// TIA Portal V16 export
// export: Created 2022-02-11T10:36:49.9262593Z, ExportSetting WithDefaults, DisplayName Totally Integrated Automation Portal, DisplayVersion V16 Update 5, DisplayName TIA Portal Version Control Interface, DisplayVersion V16 Update 2, DisplayName TIA Portal Openness, DisplayVersion V16 Update 5, DisplayName STEP 7 Professional, DisplayVersion V16 Update 5, DisplayName STEP 7 Safety, DisplayVersion V16, DisplayName WinCC Professional, DisplayVersion V16 Update 5, DisplayName SIMATIC Visualization Architect, DisplayVersion V16
FUNCTION_BLOCK "fbObjMotor_KM"   // FB9202, LAD
{ S7_Optimized_Access := 'TRUE' }
VERSION : 0.1
// stored: AutoNumber false, IsIECCheckEnabled false, IsRetainMemResEnabled false, MemoryReserve 0, SetENOAutomatically false, UDAEnableTagReadback false
   VAR_INPUT
      aMarxaAuto : Bool := FALSE;   // Activar element mode automatic
      eErrorProteccio : Bool;   // Entrada error proteccio motor filtre
      eConfirmacioMarxa : Bool;   // Senyal confirmacio marxa filtre
      bCM_Marxa : Bool := TRUE;   // Condicions necesaries activar element
      tAla_ConMar : Time := t#3s;   // Temps retard activacio alarma confirmacio marxa
      tAla_CM_Marxa : Time := t#2s;   // Temps retard activacio alarma condicions moviment
      psEnaAutoGrl : "boto";
      psEnaManualGrl : "boto";
      psAnuConMov : Bool;
      psResetAlarma : Bool;
      mFirstScan : Bool;
      "Clock_0.5Hz" : Bool;
      bSysOk : Bool := FALSE;
   END_VAR
   VAR_OUTPUT
      aMarxa : Bool;   // Sortida activacio Filtre
      be_Marxa : Bool;   // Bit estat Marxa (Confirmacio + Proteccio + Sortida)
      be_Parat : Bool;
      al_Proteccio : Bool;   // Alarma proteccio motor
      al_CM_Marxa : Bool;   // Alarma condicions moviment obrir
      al_Marxa : Bool;   // Alarma confirmacio marxa filtre
   END_VAR
   VAR
      psManMarxa : Bool;
      be_Marxa_Err : Bool;   // Error en validacio Confirmacio Marxa. Sense retard per alarma.
      bErrorCM : Bool;   // Error CM. Si activem sortida i no es compleixen les CM. Sense retard
      timAla_CM_Marxa { S7_SetPoint := 'True'} : IEC_TIMER;   // Timer retard alarma condicions moviment
      timAla_Marxa { S7_SetPoint := 'True'} : IEC_TIMER;   // Timer retard alarma marxa filtre
      bCM_Ok { S7_SetPoint := 'True'} : Bool;
      aMarxaSenseTestCM : Bool;   // Bit activacio sortida sense tenir en compte condicions moviment
      mAuxTimer : Bool;   // Bit auxiliarInicialitzacio timers
      HMI : "HMI_oMotor";
      bLast_Alarmes { S7_SetPoint := 'True'} : Bool;
   END_VAR
   VAR_TEMP
      ModeManual : Bool;
      ModeAutomatic : Bool;
      ResetAlarmes : Bool;
   END_VAR
   VAR CONSTANT
      STATUS_OBJ_ERR : Int := 10;
      STATUS_OBJ_WARNING : Int := 11;
      STATUS_OBJ_ON : Int := 1;
      STATUS_OBJ_OFF : Int := 0;
      STATUS_OBJ_UNKNOWN : Int := -1;
   END_VAR
   VAR_TEMP   // added for the SCL form of the ladder/FBD networks
      _w1 : Bool;
   END_VAR
BEGIN

REGION Network 1 (SCL): Descripció
   // Motor activat per Rele, amb confirmacio i proteccio.
END_REGION

REGION Network 2: Test habilitació mode manual. Desactivar si no tenim habilitació manual.
   // psEnaManualGrl : és el pulsador de manual de Appinfo. Si aquest està activar tots els objectes del cicle es troben en Mode Manual.
   // 
   // HMI.psEnaManual : és el pulsador de manual únic de l'objecte. Significa que la resta d'objectes es trobaràn en automàtic menys aquest.
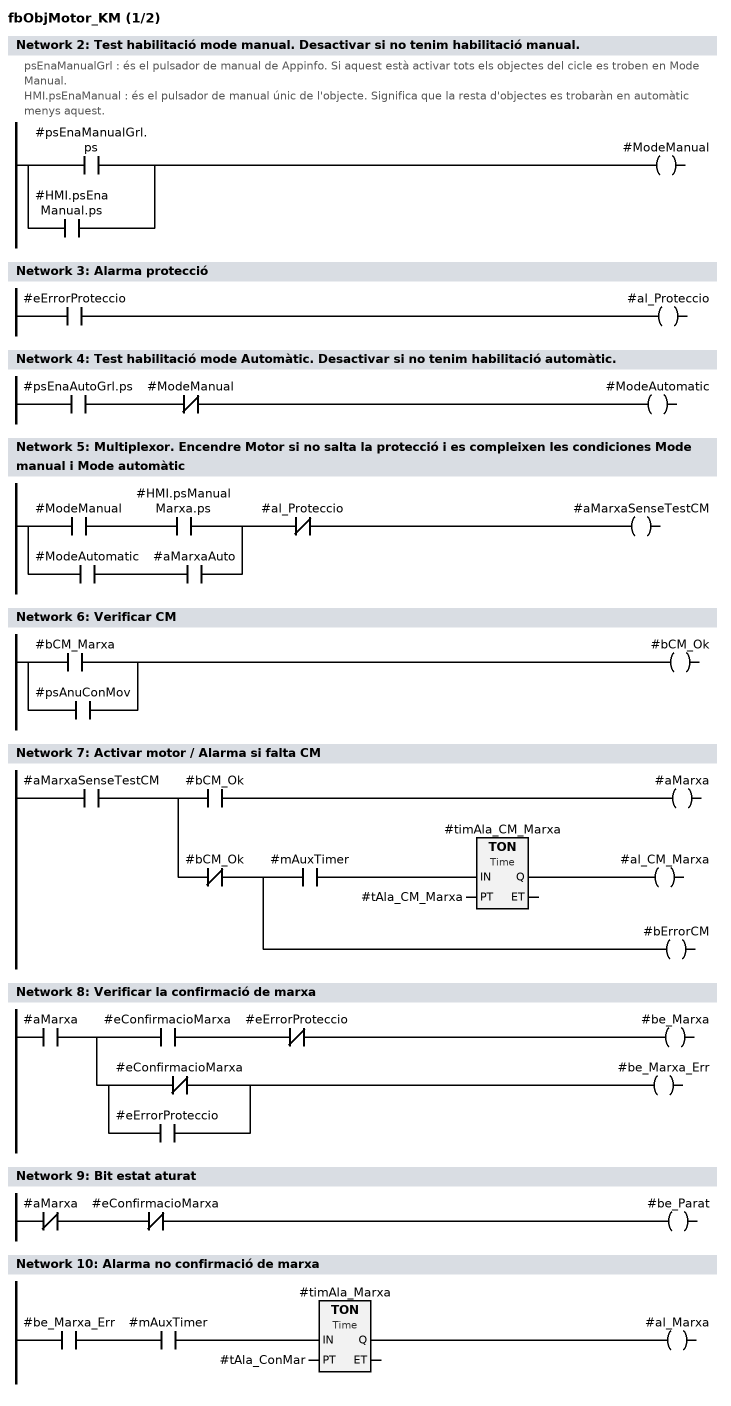
   RUNG wire#powerrail
      Contact( #psEnaManualGrl.ps )
      wire#w1
      Coil( #ModeManual )
   END_RUNG
   RUNG wire#powerrail
      Contact( #HMI.psEnaManual.ps )
   END_RUNG wire#w1
   // the same network as SCL:
   #ModeManual := #psEnaManualGrl.ps OR #HMI.psEnaManual.ps;
END_REGION

REGION Network 3: Alarma protecció
   RUNG wire#powerrail
      Contact( #eErrorProteccio )
      Coil( #al_Proteccio )
   END_RUNG
   // the same network as SCL:
   #al_Proteccio := #eErrorProteccio;
END_REGION

REGION Network 4: Test habilitació mode Automàtic. Desactivar si no tenim habilitació automàtic.
   RUNG wire#powerrail
      Contact( #psEnaAutoGrl.ps )
      I_Contact( #ModeManual )
      Coil( #ModeAutomatic )
   END_RUNG
   // the same network as SCL:
   #ModeAutomatic := #psEnaAutoGrl.ps AND NOT #ModeManual;
END_REGION

REGION Network 5: Multiplexor. Encendre Motor si no salta la protecció i es compleixen les condiciones Mode manual i Mode automàtic
   RUNG wire#powerrail
      Contact( #ModeManual )
      Contact( #HMI.psManualMarxa.ps )
      wire#w1
      I_Contact( #al_Proteccio )
      Coil( #aMarxaSenseTestCM )
   END_RUNG
   RUNG wire#powerrail
      Contact( #ModeAutomatic )
      Contact( #aMarxaAuto )
   END_RUNG wire#w1
   // the same network as SCL:
   #aMarxaSenseTestCM := ((#ModeManual AND #HMI.psManualMarxa.ps) OR (#ModeAutomatic AND #aMarxaAuto)) AND NOT #al_Proteccio;
END_REGION

REGION Network 6: Verificar CM
   RUNG wire#powerrail
      Contact( #bCM_Marxa )
      wire#w1
      Coil( #bCM_Ok )
   END_RUNG
   RUNG wire#powerrail
      Contact( #psAnuConMov )
   END_RUNG wire#w1
   // the same network as SCL:
   #bCM_Ok := #bCM_Marxa OR #psAnuConMov;
END_REGION

REGION Network 7: Activar motor / Alarma si falta CM
   RUNG wire#powerrail
      Contact( #aMarxaSenseTestCM )
      wire#w1
      Contact( #bCM_Ok )
      Coil( #aMarxa )
   END_RUNG
   RUNG wire#w1
      I_Contact( #bCM_Ok )
      wire#w2
      Contact( #mAuxTimer )
      { S7_Templates := "time_type := Time" } #timAla_CM_Marxa.TON(pt := #tAla_CM_Marxa, et =>)
      Coil( #al_CM_Marxa )
   END_RUNG
   RUNG wire#w2
      Coil( #bErrorCM )
   END_RUNG
   // the same network as SCL:
   #aMarxa := #aMarxaSenseTestCM AND #bCM_Ok;
   #_w1 := #aMarxaSenseTestCM AND NOT #bCM_Ok;
   #timAla_CM_Marxa.TON(IN := #_w1 AND #mAuxTimer, PT := #tAla_CM_Marxa);
   #al_CM_Marxa := #timAla_CM_Marxa.Q;
   #bErrorCM := #_w1;
END_REGION

REGION Network 8: Verificar la confirmació de marxa
   RUNG wire#powerrail
      Contact( #aMarxa )
      wire#w1
      Contact( #eConfirmacioMarxa )
      I_Contact( #eErrorProteccio )
      Coil( #be_Marxa )
   END_RUNG
   RUNG wire#w1
      I_Contact( #eConfirmacioMarxa )
      wire#w2
      Coil( #be_Marxa_Err )
   END_RUNG
   RUNG wire#w1
      Contact( #eErrorProteccio )
   END_RUNG wire#w2
   // the same network as SCL:
   #be_Marxa := #aMarxa AND #eConfirmacioMarxa AND NOT #eErrorProteccio;
   #be_Marxa_Err := #aMarxa AND (NOT #eConfirmacioMarxa OR #eErrorProteccio);
END_REGION

REGION Network 9: Bit estat aturat
   RUNG wire#powerrail
      I_Contact( #aMarxa )
      I_Contact( #eConfirmacioMarxa )
      Coil( #be_Parat )
   END_RUNG
   // the same network as SCL:
   #be_Parat := NOT #aMarxa AND NOT #eConfirmacioMarxa;
END_REGION

REGION Network 10: Alarma no confirmació de marxa
   RUNG wire#powerrail
      Contact( #be_Marxa_Err )
      Contact( #mAuxTimer )
      { S7_Templates := "time_type := Time" } #timAla_Marxa.TON(pt := #tAla_ConMar, et =>)
      Coil( #al_Marxa )
   END_RUNG
   // the same network as SCL:
   #timAla_Marxa.TON(IN := #be_Marxa_Err AND #mAuxTimer, PT := #tAla_ConMar);
   #al_Marxa := #timAla_Marxa.Q;
END_REGION

REGION Network 11: Verificar pulsació alarmes
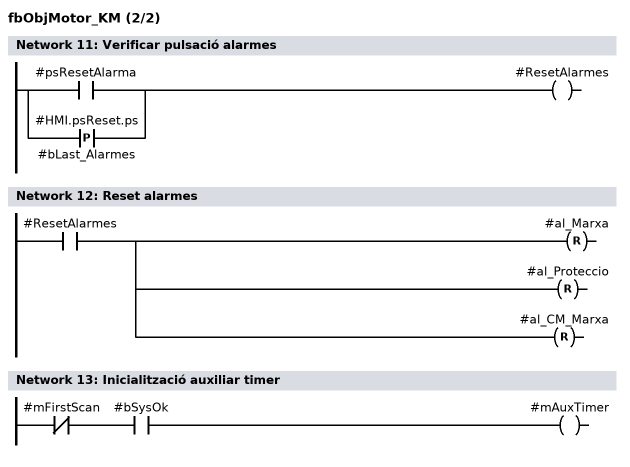
   RUNG wire#powerrail
      Contact( #psResetAlarma )
      wire#w1
      Coil( #ResetAlarmes )
   END_RUNG
   RUNG wire#powerrail
      P_Contact(operand := #HMI.psReset.ps, bit := #bLast_Alarmes)
   END_RUNG wire#w1
   // the same network as SCL:
   #_w1 := #HMI.psReset.ps AND NOT #bLast_Alarmes;   // rising edge of #HMI.psReset.ps
   #bLast_Alarmes := #HMI.psReset.ps;
   #ResetAlarmes := #psResetAlarma OR #_w1;
END_REGION

REGION Network 12: Reset alarmes
   RUNG wire#powerrail
      Contact( #ResetAlarmes )
      wire#w1
      R_Coil( #al_Marxa )
   END_RUNG
   RUNG wire#w1
      R_Coil( #al_Proteccio )
   END_RUNG
   RUNG wire#w1
      R_Coil( #al_CM_Marxa )
   END_RUNG
   // the same network as SCL:
   IF #ResetAlarmes THEN
       #al_Marxa := FALSE;
       #al_Proteccio := FALSE;
       #al_CM_Marxa := FALSE;
   END_IF;
END_REGION

REGION Network 13: Inicialització auxiliar timer
   RUNG wire#powerrail
      I_Contact( #mFirstScan )
      Contact( #bSysOk )
      Coil( #mAuxTimer )
   END_RUNG
   // the same network as SCL:
   #mAuxTimer := NOT #mFirstScan AND #bSysOk;
END_REGION

REGION Network 14 (SCL): HMI estat Motor
       IF (#al_Marxa OR #al_CM_Marxa OR #eErrorProteccio) THEN
           #HMI.iStatusDisplay := #STATUS_OBJ_ERR;                // Error = 10
           #HMI.bDisplayError := TRUE;
           #HMI.bDisplayWarning := FALSE;
           #HMI.bDisplayOk := FALSE;

       ELSIF (#be_Marxa_Err OR #bErrorCM) THEN
           #HMI.iStatusDisplay := #STATUS_OBJ_WARNING;            // Warning = 11
           #HMI.bDisplayError := FALSE;
           #HMI.bDisplayWarning := TRUE;
           #HMI.bDisplayOk := FALSE;

       ELSIF #be_Marxa THEN
           #HMI.iStatusDisplay := #STATUS_OBJ_ON;                 // Bit estat Marxa Auto = 1
           #HMI.bDisplayError := FALSE;
           #HMI.bDisplayWarning := FALSE;
           #HMI.bDisplayOk := TRUE;

       ELSIF #be_Parat THEN
           #HMI.iStatusDisplay := #STATUS_OBJ_OFF;                 // Bit estat Marxa Auto = 1
           #HMI.bDisplayError := FALSE;
           #HMI.bDisplayWarning := FALSE;
           #HMI.bDisplayOk := TRUE;

       ELSIF #aMarxa THEN
           IF #"Clock_0.5Hz" THEN
               #HMI.iStatusDisplay := #STATUS_OBJ_WARNING;
           ELSE
               #HMI.iStatusDisplay := #STATUS_OBJ_ON;
           END_IF;
           #HMI.bDisplayError := FALSE;
           #HMI.bDisplayWarning := TRUE;
           #HMI.bDisplayOk := FALSE;

       ELSE
           IF #"Clock_0.5Hz" THEN
               #HMI.iStatusDisplay := #STATUS_OBJ_WARNING;
           ELSE
               #HMI.iStatusDisplay := #STATUS_OBJ_OFF;
           END_IF;
           #HMI.bDisplayError := FALSE;
           #HMI.bDisplayWarning := TRUE;
           #HMI.bDisplayOk := FALSE;

       END_IF;
END_REGION
END_FUNCTION_BLOCK
